// TIA Portal V20 export
TYPE "LKinCtrl_typeMoveDirectParameter"
   STRUCT
      linkConstellation : DWord := 16#FFFF_FFFF;   // linkConstellation (effective for MoveDirect commands only)
      positionMode : DInt := 1;   // 1: absolute cartesian position and absolute orientation; 2: absolute cartesian position and relative orientation (effective for MoveDirect commands only)
      turnJoint : Array[1..6] of DInt;   // turn joint setting (effective for MoveDirect commands only)
   END_STRUCT;
END_TYPE
